FUNCTION_BLOCK E_CTUD_UDINT (* Event-Driven Up-Down Counter *)
  (* Standard: 61499-1-A.x; Classification: Event-driven blocks; Function: Up-Down-counter; Description: Copyright (c) 2017, 2024 fortiss GmbH, JKU, HR Agrartechnik GmbH This program and the accompanying materials are made available under the terms of the Eclipse Public License 2.0 which is available at https://www.eclipse.org/legal/epl-2.0/ SPDX-License-Identifier: EPL-2.0 *)
  (* Version 1.0, 2017-09-22, Alois Zoitl, fortiss GmbH, initial API and implementation and/or initial documentation (E_CTUD) *)
  (* Version 1.1, 2019-07-09, Alois Zoitl, JKU, fixed bug in down counting (E_CTUD) *)
  (* Version 1.2, 2024-02-10, Franz Höpfinger, HR Agrartechnik GmbH, Copy over E_CTUD to E_CTUD_UDINT *)
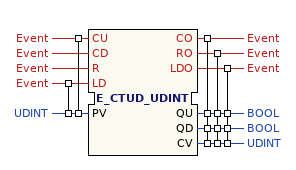
  EVENT_INPUT
    CU WITH PV; (* Count Up *)
    CD; (* Count Down *)
    R; (* Reset *)
    LD WITH PV; (* Load *)
  END_EVENT
  EVENT_OUTPUT
    CO WITH QU, CV, QD; (* Count Output Event *)
    RO WITH QU, CV, QD; (* Reset Output Event *)
    LDO WITH QU, QD, CV;
  END_EVENT
  VAR_INPUT
    PV : UDINT; (* Preset Value *)
  END_VAR
  VAR_OUTPUT
    QU : BOOL; (* CV &gt;=PV *)
    QD : BOOL; (* CV &lt;= 0 *)
    CV : UDINT; (* Counter Value *)
  END_VAR
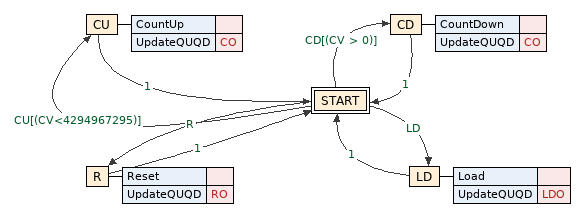
  EC_STATES
    START;
    CU : CountUp, UpdateQUQD -> CO;
    R : Reset, UpdateQUQD -> RO;
    CD : CountDown, UpdateQUQD -> CO;
    LD : Load, UpdateQUQD -> LDO;
  END_STATES
  EC_TRANSITIONS
    START TO CU := CU[(CV<4294967295)];
    CU TO START := 1;
    START TO R := R;
    R TO START := 1;
    START TO CD := CD[(CV > 0)];
    CD TO START := 1;
    START TO LD := LD;
    LD TO START := 1;
  END_TRANSITIONS
  ALGORITHM CountUp IN ST:
CV := CV + 1;
  END_ALGORITHM
  ALGORITHM Reset IN ST:
CV := 0;
  END_ALGORITHM
  ALGORITHM Load IN ST:
CV := PV;
  END_ALGORITHM
  ALGORITHM UpdateQUQD IN ST:
QU := (CV >= PV);
QD := (CV = 0);
  END_ALGORITHM
  ALGORITHM CountDown IN ST:
CV := CV - 1;
  END_ALGORITHM
END_FUNCTION_BLOCK
